(* IEC 61131-3 sources: verifaps-lib/geteta/examples/RTT_if (part 5) *)

        Pusher_states_t#Reset_interconnect_Slide1_Black:
             b_Pusher$_transit  := FALSE;
             b_Pusher$interconnect3  := FALSE;
             b_Pusher$Timer3$IN  := FALSE;
             b_Pusher$Timer3$PT  := USINT#0;
            IF  b_Pusher$Timer3$IN  THEN
                 b_Pusher$Timer3$Q  := ( b_Pusher$Timer3$ET  = USINT#0);
                IF ( b_Pusher$Timer3$ET  > USINT#0) THEN
                     b_Pusher$Timer3$ET  := ( b_Pusher$Timer3$ET  - USINT#1);
                ELSE
                     b_Pusher$Timer3$ET  := USINT#0;
                END_IF
            ELSE
                 b_Pusher$Timer3$Q  := FALSE;
                 b_Pusher$Timer3$ET  :=  b_Pusher$Timer3$PT ;
            END_IF
             b_Pusher$interconnect_Slide1_Black  := FALSE;
             b_Pusher$Timer_Slide1_Black$IN  := FALSE;
             b_Pusher$Timer_Slide1_Black$PT  := USINT#0;
            IF  b_Pusher$Timer_Slide1_Black$IN  THEN
                 b_Pusher$Timer_Slide1_Black$Q  := ( b_Pusher$Timer_Slide1_Black$ET  = USINT#0);
                IF ( b_Pusher$Timer_Slide1_Black$ET  > USINT#0) THEN
                     b_Pusher$Timer_Slide1_Black$ET  := ( b_Pusher$Timer_Slide1_Black$ET  - USINT#1);
                ELSE
                     b_Pusher$Timer_Slide1_Black$ET  := USINT#0;
                END_IF
            ELSE
                 b_Pusher$Timer_Slide1_Black$Q  := FALSE;
                 b_Pusher$Timer_Slide1_Black$ET  :=  b_Pusher$Timer_Slide1_Black$PT ;
            END_IF
             b_Pusher$Slide1_black  := ( b_Pusher$Slide1_black  - INT#1);
             b_Pusher$Priority_Var_Black  := ( b_Pusher$Priority_Var_Black  - INT#1);
            IF TRUE THEN
                 b_Pusher$_transit  := TRUE;
                 b_Pusher$_state  := Pusher_states_t#Interstep_2;
            END_IF

        Pusher_states_t#Reset_interconnect_Slide1_Metal:
             b_Pusher$_transit  := FALSE;
             b_Pusher$interconnect3  := FALSE;
             b_Pusher$Timer3$IN  := FALSE;
             b_Pusher$Timer3$PT  := USINT#0;
            IF  b_Pusher$Timer3$IN  THEN
                 b_Pusher$Timer3$Q  := ( b_Pusher$Timer3$ET  = USINT#0);
                IF ( b_Pusher$Timer3$ET  > USINT#0) THEN
                     b_Pusher$Timer3$ET  := ( b_Pusher$Timer3$ET  - USINT#1);
                ELSE
                     b_Pusher$Timer3$ET  := USINT#0;
                END_IF
            ELSE
                 b_Pusher$Timer3$Q  := FALSE;
                 b_Pusher$Timer3$ET  :=  b_Pusher$Timer3$PT ;
            END_IF
             b_Pusher$interconnect_Slide1_Metal  := FALSE;
             b_Pusher$Timer_Slide1_Metal$IN  := FALSE;
             b_Pusher$Timer_Slide1_Metal$PT  := USINT#0;
            IF  b_Pusher$Timer_Slide1_Metal$IN  THEN
                 b_Pusher$Timer_Slide1_Metal$Q  := ( b_Pusher$Timer_Slide1_Metal$ET  = USINT#0);
                IF ( b_Pusher$Timer_Slide1_Metal$ET  > USINT#0) THEN
                     b_Pusher$Timer_Slide1_Metal$ET  := ( b_Pusher$Timer_Slide1_Metal$ET  - USINT#1);
                ELSE
                     b_Pusher$Timer_Slide1_Metal$ET  := USINT#0;
                END_IF
            ELSE
                 b_Pusher$Timer_Slide1_Metal$Q  := FALSE;
                 b_Pusher$Timer_Slide1_Metal$ET  :=  b_Pusher$Timer_Slide1_Metal$PT ;
            END_IF
             b_Pusher$Slide1_metal  := ( b_Pusher$Slide1_metal  - INT#1);
             b_Pusher$Priority_Var_Metal  := ( b_Pusher$Priority_Var_Metal  - INT#1);
            IF TRUE THEN
                 b_Pusher$_transit  := TRUE;
                 b_Pusher$_state  := Pusher_states_t#Interstep_2;
            END_IF

        Pusher_states_t#Reset_interconnect_Slide1_White:
             b_Pusher$_transit  := FALSE;
             b_Pusher$interconnect3  := FALSE;
             b_Pusher$Timer3$IN  := FALSE;
             b_Pusher$Timer3$PT  := USINT#0;
            IF  b_Pusher$Timer3$IN  THEN
                 b_Pusher$Timer3$Q  := ( b_Pusher$Timer3$ET  = USINT#0);
                IF ( b_Pusher$Timer3$ET  > USINT#0) THEN
                     b_Pusher$Timer3$ET  := ( b_Pusher$Timer3$ET  - USINT#1);
                ELSE
                     b_Pusher$Timer3$ET  := USINT#0;
                END_IF
            ELSE
                 b_Pusher$Timer3$Q  := FALSE;
                 b_Pusher$Timer3$ET  :=  b_Pusher$Timer3$PT ;
            END_IF
             b_Pusher$interconnect_Slide1_White  := FALSE;
             b_Pusher$Timer_Slide1_White$IN  := FALSE;
             b_Pusher$Timer_Slide1_White$PT  := USINT#0;
            IF  b_Pusher$Timer_Slide1_White$IN  THEN
                 b_Pusher$Timer_Slide1_White$Q  := ( b_Pusher$Timer_Slide1_White$ET  = USINT#0);
                IF ( b_Pusher$Timer_Slide1_White$ET  > USINT#0) THEN
                     b_Pusher$Timer_Slide1_White$ET  := ( b_Pusher$Timer_Slide1_White$ET  - USINT#1);
                ELSE
                     b_Pusher$Timer_Slide1_White$ET  := USINT#0;
                END_IF
            ELSE
                 b_Pusher$Timer_Slide1_White$Q  := FALSE;
                 b_Pusher$Timer_Slide1_White$ET  :=  b_Pusher$Timer_Slide1_White$PT ;
            END_IF
             b_Pusher$Slide1_white  := ( b_Pusher$Slide1_white  - INT#1);
             b_Pusher$Priority_Var_White  := ( b_Pusher$Priority_Var_White  - INT#1);
            IF TRUE THEN
                 b_Pusher$_transit  := TRUE;
                 b_Pusher$_state  := Pusher_states_t#Interstep_2;
            END_IF

        Pusher_states_t#Reset_interconnect_Slide2_Black:
             b_Pusher$_transit  := FALSE;
             b_Pusher$interconnect3  := FALSE;
             b_Pusher$Timer3$IN  := FALSE;
             b_Pusher$Timer3$PT  := USINT#0;
            IF  b_Pusher$Timer3$IN  THEN
                 b_Pusher$Timer3$Q  := ( b_Pusher$Timer3$ET  = USINT#0);
                IF ( b_Pusher$Timer3$ET  > USINT#0) THEN
                     b_Pusher$Timer3$ET  := ( b_Pusher$Timer3$ET  - USINT#1);
                ELSE
                     b_Pusher$Timer3$ET  := USINT#0;
                END_IF
            ELSE
                 b_Pusher$Timer3$Q  := FALSE;
                 b_Pusher$Timer3$ET  :=  b_Pusher$Timer3$PT ;
            END_IF
             b_Pusher$interconnect_Slide2_Black  := FALSE;
             b_Pusher$Timer_Slide2_Black$IN  := FALSE;
             b_Pusher$Timer_Slide2_Black$PT  := USINT#0;
            IF  b_Pusher$Timer_Slide2_Black$IN  THEN
                 b_Pusher$Timer_Slide2_Black$Q  := ( b_Pusher$Timer_Slide2_Black$ET  = USINT#0);
                IF ( b_Pusher$Timer_Slide2_Black$ET  > USINT#0) THEN
                     b_Pusher$Timer_Slide2_Black$ET  := ( b_Pusher$Timer_Slide2_Black$ET  - USINT#1);
                ELSE
                     b_Pusher$Timer_Slide2_Black$ET  := USINT#0;
                END_IF
            ELSE
                 b_Pusher$Timer_Slide2_Black$Q  := FALSE;
                 b_Pusher$Timer_Slide2_Black$ET  :=  b_Pusher$Timer_Slide2_Black$PT ;
            END_IF
             b_Pusher$Slide2_black  := ( b_Pusher$Slide2_black  - INT#1);
             b_Pusher$Priority_Var_Black  := ( b_Pusher$Priority_Var_Black  - INT#1);
            IF TRUE THEN
                 b_Pusher$_transit  := TRUE;
                 b_Pusher$_state  := Pusher_states_t#Interstep_2;
            END_IF

        Pusher_states_t#Reset_interconnect_Slide2_Metal:
             b_Pusher$_transit  := FALSE;
             b_Pusher$interconnect3  := FALSE;
             b_Pusher$Timer3$IN  := FALSE;
             b_Pusher$Timer3$PT  := USINT#0;
            IF  b_Pusher$Timer3$IN  THEN
                 b_Pusher$Timer3$Q  := ( b_Pusher$Timer3$ET  = USINT#0);
                IF ( b_Pusher$Timer3$ET  > USINT#0) THEN
                     b_Pusher$Timer3$ET  := ( b_Pusher$Timer3$ET  - USINT#1);
                ELSE
                     b_Pusher$Timer3$ET  := USINT#0;
                END_IF
            ELSE
                 b_Pusher$Timer3$Q  := FALSE;
                 b_Pusher$Timer3$ET  :=  b_Pusher$Timer3$PT ;
            END_IF
             b_Pusher$interconnect_Slide2_Metal  := FALSE;
             b_Pusher$Timer_Slide2_Metal$IN  := FALSE;
             b_Pusher$Timer_Slide2_Metal$PT  := USINT#0;
            IF  b_Pusher$Timer_Slide2_Metal$IN  THEN
                 b_Pusher$Timer_Slide2_Metal$Q  := ( b_Pusher$Timer_Slide2_Metal$ET  = USINT#0);
                IF ( b_Pusher$Timer_Slide2_Metal$ET  > USINT#0) THEN
                     b_Pusher$Timer_Slide2_Metal$ET  := ( b_Pusher$Timer_Slide2_Metal$ET  - USINT#1);
                ELSE
                     b_Pusher$Timer_Slide2_Metal$ET  := USINT#0;
                END_IF
            ELSE
                 b_Pusher$Timer_Slide2_Metal$Q  := FALSE;
                 b_Pusher$Timer_Slide2_Metal$ET  :=  b_Pusher$Timer_Slide2_Metal$PT ;
            END_IF
             b_Pusher$Slide2_metal  := ( b_Pusher$Slide2_metal  - INT#1);
             b_Pusher$Priority_Var_Metal  := ( b_Pusher$Priority_Var_Metal  - INT#1);
            IF TRUE THEN
                 b_Pusher$_transit  := TRUE;
                 b_Pusher$_state  := Pusher_states_t#Interstep_2;
            END_IF

        Pusher_states_t#Reset_interconnect_Slide2_White:
             b_Pusher$_transit  := FALSE;
             b_Pusher$interconnect3  := FALSE;
             b_Pusher$Timer3$IN  := FALSE;
             b_Pusher$Timer3$PT  := USINT#0;
            IF  b_Pusher$Timer3$IN  THEN
                 b_Pusher$Timer3$Q  := ( b_Pusher$Timer3$ET  = USINT#0);
                IF ( b_Pusher$Timer3$ET  > USINT#0) THEN
                     b_Pusher$Timer3$ET  := ( b_Pusher$Timer3$ET  - USINT#1);
                ELSE
                     b_Pusher$Timer3$ET  := USINT#0;
                END_IF
            ELSE
                 b_Pusher$Timer3$Q  := FALSE;
                 b_Pusher$Timer3$ET  :=  b_Pusher$Timer3$PT ;
            END_IF
             b_Pusher$interconnect_Slide2_White  := FALSE;
             b_Pusher$Timer_Slide2_White$IN  := FALSE;
             b_Pusher$Timer_Slide2_White$PT  := USINT#0;
            IF  b_Pusher$Timer_Slide2_White$IN  THEN
                 b_Pusher$Timer_Slide2_White$Q  := ( b_Pusher$Timer_Slide2_White$ET  = USINT#0);
                IF ( b_Pusher$Timer_Slide2_White$ET  > USINT#0) THEN
                     b_Pusher$Timer_Slide2_White$ET  := ( b_Pusher$Timer_Slide2_White$ET  - USINT#1);
                ELSE
                     b_Pusher$Timer_Slide2_White$ET  := USINT#0;
                END_IF
            ELSE
                 b_Pusher$Timer_Slide2_White$Q  := FALSE;
                 b_Pusher$Timer_Slide2_White$ET  :=  b_Pusher$Timer_Slide2_White$PT ;
            END_IF
             b_Pusher$Slide2_white  := ( b_Pusher$Slide2_white  - INT#1);
             b_Pusher$Priority_Var_White  := ( b_Pusher$Priority_Var_White  - INT#1);
            IF TRUE THEN
                 b_Pusher$_transit  := TRUE;
                 b_Pusher$_state  := Pusher_states_t#Interstep_2;
            END_IF

        Pusher_states_t#Reset_interconnect_Slide3_Metal:
             b_Pusher$_transit  := FALSE;
             b_Pusher$interconnect3  := FALSE;
             b_Pusher$Timer3$IN  := FALSE;
             b_Pusher$Timer3$PT  := USINT#0;
            IF  b_Pusher$Timer3$IN  THEN
                 b_Pusher$Timer3$Q  := ( b_Pusher$Timer3$ET  = USINT#0);
                IF ( b_Pusher$Timer3$ET  > USINT#0) THEN
                     b_Pusher$Timer3$ET  := ( b_Pusher$Timer3$ET  - USINT#1);
                ELSE
                     b_Pusher$Timer3$ET  := USINT#0;
                END_IF
            ELSE
                 b_Pusher$Timer3$Q  := FALSE;
                 b_Pusher$Timer3$ET  :=  b_Pusher$Timer3$PT ;
            END_IF
             b_Pusher$Slide3_metal  := ( b_Pusher$Slide3_metal  - INT#1);
             b_Pusher$Priority_Var_Metal  := ( b_Pusher$Priority_Var_Metal  - INT#1);
            IF TRUE THEN
                 b_Pusher$_transit  := TRUE;
                 b_Pusher$_state  := Pusher_states_t#Interstep_2;
            END_IF

        Pusher_states_t#Reset_interconnect_Slide3_White:
             b_Pusher$_transit  := FALSE;
             b_Pusher$interconnect3  := FALSE;
             b_Pusher$Timer3$IN  := FALSE;
             b_Pusher$Timer3$PT  := USINT#0;
            IF  b_Pusher$Timer3$IN  THEN
                 b_Pusher$Timer3$Q  := ( b_Pusher$Timer3$ET  = USINT#0);
                IF ( b_Pusher$Timer3$ET  > USINT#0) THEN
                     b_Pusher$Timer3$ET  := ( b_Pusher$Timer3$ET  - USINT#1);
                ELSE
                     b_Pusher$Timer3$ET  := USINT#0;
                END_IF
            ELSE
                 b_Pusher$Timer3$Q  := FALSE;
                 b_Pusher$Timer3$ET  :=  b_Pusher$Timer3$PT ;
            END_IF
             b_Pusher$Slide3_white  := ( b_Pusher$Slide3_white  - INT#1);
             b_Pusher$Priority_Var_White  := ( b_Pusher$Priority_Var_White  - INT#1);
            IF TRUE THEN
                 b_Pusher$_transit  := TRUE;
                 b_Pusher$_state  := Pusher_states_t#Interstep_2;
            END_IF

        Pusher_states_t#Second_Slide_Timer_Black:
             b_Pusher$_transit  := FALSE;
            IF ( b_Pusher$SorterLightnesssensorCraneInterfaceInverse  = TRUE) THEN
                 b_Pusher$Timer_Slide2_Black$IN  :=  b_Pusher$SorterLightnesssensorCraneInterfaceInverse ;
                 b_Pusher$Timer_Slide2_Black$PT  :=  b_Pusher$Duration_Slide2_Black ;
                IF  b_Pusher$Timer_Slide2_Black$IN  THEN
                     b_Pusher$Timer_Slide2_Black$Q  := ( b_Pusher$Timer_Slide2_Black$ET  = USINT#0);
                    IF ( b_Pusher$Timer_Slide2_Black$ET  > USINT#0) THEN
                         b_Pusher$Timer_Slide2_Black$ET  := ( b_Pusher$Timer_Slide2_Black$ET  - USINT#1);
                    ELSE
                         b_Pusher$Timer_Slide2_Black$ET  := USINT#0;
                    END_IF
                ELSE
                     b_Pusher$Timer_Slide2_Black$Q  := FALSE;
                     b_Pusher$Timer_Slide2_Black$ET  :=  b_Pusher$Timer_Slide2_Black$PT ;
                END_IF
                 b_Pusher$interconnect_Slide2_Black  :=  b_Pusher$Timer_Slide2_Black$Q ;
            END_IF
            IF  b_Pusher$interconnect_Slide2_Black  THEN
                 b_Pusher$_transit  := TRUE;
                 b_Pusher$_state  := Pusher_states_t#PusherY2_Move_Out_Black;
            END_IF

        Pusher_states_t#Second_Slide_Timer_Metal:
             b_Pusher$_transit  := FALSE;
             b_Pusher$Timer_Slide2_Metal$IN  := TRUE;
             b_Pusher$Timer_Slide2_Metal$PT  :=  b_Pusher$Duration_Slide2_Metal ;
            IF  b_Pusher$Timer_Slide2_Metal$IN  THEN
                 b_Pusher$Timer_Slide2_Metal$Q  := ( b_Pusher$Timer_Slide2_Metal$ET  = USINT#0);
                IF ( b_Pusher$Timer_Slide2_Metal$ET  > USINT#0) THEN
                     b_Pusher$Timer_Slide2_Metal$ET  := ( b_Pusher$Timer_Slide2_Metal$ET  - USINT#1);
                ELSE
                     b_Pusher$Timer_Slide2_Metal$ET  := USINT#0;
                END_IF
            ELSE
                 b_Pusher$Timer_Slide2_Metal$Q  := FALSE;
                 b_Pusher$Timer_Slide2_Metal$ET  :=  b_Pusher$Timer_Slide2_Metal$PT ;
            END_IF
             b_Pusher$interconnect_Slide2_Metal  :=  b_Pusher$Timer_Slide2_Metal$Q ;
            IF  b_Pusher$interconnect_Slide2_Metal  THEN
                 b_Pusher$_transit  := TRUE;
                 b_Pusher$_state  := Pusher_states_t#PusherY2_Move_Out_Metal;
            END_IF

        Pusher_states_t#Second_Slide_Timer_White:
             b_Pusher$_transit  := FALSE;
             b_Pusher$Timer_Slide2_White$IN  := TRUE;
             b_Pusher$Timer_Slide2_White$PT  :=  b_Pusher$Duration_Slide2_White ;
            IF  b_Pusher$Timer_Slide2_White$IN  THEN
                 b_Pusher$Timer_Slide2_White$Q  := ( b_Pusher$Timer_Slide2_White$ET  = USINT#0);
                IF ( b_Pusher$Timer_Slide2_White$ET  > USINT#0) THEN
                     b_Pusher$Timer_Slide2_White$ET  := ( b_Pusher$Timer_Slide2_White$ET  - USINT#1);
                ELSE
                     b_Pusher$Timer_Slide2_White$ET  := USINT#0;
                END_IF
            ELSE
                 b_Pusher$Timer_Slide2_White$Q  := FALSE;
                 b_Pusher$Timer_Slide2_White$ET  :=  b_Pusher$Timer_Slide2_White$PT ;
            END_IF
             b_Pusher$interconnect_Slide2_White  :=  b_Pusher$Timer_Slide2_White$Q ;
            IF  b_Pusher$interconnect_Slide2_White  THEN
                 b_Pusher$_transit  := TRUE;
                 b_Pusher$_state  := Pusher_states_t#PusherY2_Move_Out_White;
            END_IF

        Pusher_states_t#Second_Slide_black_workpieces:
             b_Pusher$_transit  := FALSE;
            IF TRUE THEN
                 b_Pusher$_transit  := TRUE;
                 b_Pusher$_state  := Pusher_states_t#Second_Slide_Timer_Black;
            END_IF

        Pusher_states_t#Second_Slide_metal_workpieces:
             b_Pusher$_transit  := FALSE;
            IF ( b_Pusher$SorterLightnessSensorPusher2  AND  b_Pusher$SorterCapacitiveSensorPusher2 ) THEN
                 b_Pusher$_transit  := TRUE;
                 b_Pusher$_state  := Pusher_states_t#Second_Test_For_Metal;
            END_IF

        Pusher_states_t#Second_Slide_white_workpieces:
             b_Pusher$_transit  := FALSE;
            IF ( b_Pusher$SorterLightnessSensorPusher2  AND NOT  b_Pusher$SorterCapacitiveSensorPusher2 ) THEN
                 b_Pusher$_transit  := TRUE;
                 b_Pusher$_state  := Pusher_states_t#Second_Test_For_White;
            END_IF

        Pusher_states_t#Second_Test_For_Metal:
             b_Pusher$_transit  := FALSE;
            IF TRUE THEN
                 b_Pusher$_transit  := TRUE;
                 b_Pusher$_state  := Pusher_states_t#Second_Slide_Timer_Metal;
            END_IF

        Pusher_states_t#Second_Test_For_White:
             b_Pusher$_transit  := FALSE;
            IF TRUE THEN
                 b_Pusher$_transit  := TRUE;
                 b_Pusher$_state  := Pusher_states_t#Second_Slide_Timer_White;
            END_IF

        Pusher_states_t#Third_Slide_black_workpieces:
             b_Pusher$_transit  := FALSE;
            IF (NOT  b_Pusher$SorterLightnessSensorPusher2  AND NOT  b_Pusher$SorterCapacitiveSensorPusher2 ) THEN
                 b_Pusher$_transit  := TRUE;
                 b_Pusher$_state  := Pusher_states_t#Wait_Black;
            END_IF

        Pusher_states_t#Third_Slide_metal_workpieces:
             b_Pusher$_transit  := FALSE;
            IF ( b_Pusher$SorterLightnessSensorPusher2  AND  b_Pusher$SorterCapacitiveSensorPusher2 ) THEN
                 b_Pusher$_transit  := TRUE;
                 b_Pusher$_state  := Pusher_states_t#Wait_Metal;
            END_IF

        Pusher_states_t#Third_Slide_white_workpieces:
             b_Pusher$_transit  := FALSE;
            IF ( b_Pusher$SorterLightnessSensorPusher2  AND NOT  b_Pusher$SorterCapacitiveSensorPusher2 ) THEN
                 b_Pusher$_transit  := TRUE;
                 b_Pusher$_state  := Pusher_states_t#Wait_White;
            END_IF

        Pusher_states_t#Wait_Black:
             b_Pusher$_transit  := FALSE;
            IF ((NOT  b_Pusher$SorterLightnessSensorPusher2  AND NOT  b_Pusher$SorterCapacitiveSensorPusher2 ) = TRUE) THEN
                 b_Pusher$Timer2$IN  := (NOT  b_Pusher$SorterLightnessSensorPusher2  AND NOT  b_Pusher$SorterCapacitiveSensorPusher2 );
                 b_Pusher$Timer2$PT  :=  b_Pusher$Duration2 ;
                IF  b_Pusher$Timer2$IN  THEN
                     b_Pusher$Timer2$Q  := ( b_Pusher$Timer2$ET  = USINT#0);
                    IF ( b_Pusher$Timer2$ET  > USINT#0) THEN
                         b_Pusher$Timer2$ET  := ( b_Pusher$Timer2$ET  - USINT#1);
                    ELSE
                         b_Pusher$Timer2$ET  := USINT#0;
                    END_IF
                ELSE
                     b_Pusher$Timer2$Q  := FALSE;
                     b_Pusher$Timer2$ET  :=  b_Pusher$Timer2$PT ;
                END_IF
                 b_Pusher$interconnect2  :=  b_Pusher$Timer2$Q ;
            END_IF
            IF  b_Pusher$interconnect2  THEN
                 b_Pusher$_transit  := TRUE;
                 b_Pusher$_state  := Pusher_states_t#Reset_interconnect3;
            END_IF

        Pusher_states_t#Wait_Metal:
             b_Pusher$_transit  := FALSE;
             b_Pusher$Timer3$IN  := TRUE;
             b_Pusher$Timer3$PT  :=  b_Pusher$Duration3 ;
            IF  b_Pusher$Timer3$IN  THEN
                 b_Pusher$Timer3$Q  := ( b_Pusher$Timer3$ET  = USINT#0);
                IF ( b_Pusher$Timer3$ET  > USINT#0) THEN
                     b_Pusher$Timer3$ET  := ( b_Pusher$Timer3$ET  - USINT#1);
                ELSE
                     b_Pusher$Timer3$ET  := USINT#0;
                END_IF
            ELSE
                 b_Pusher$Timer3$Q  := FALSE;
                 b_Pusher$Timer3$ET  :=  b_Pusher$Timer3$PT ;
            END_IF
             b_Pusher$interconnect3  :=  b_Pusher$Timer3$Q ;
            IF  b_Pusher$interconnect3  THEN
                 b_Pusher$_transit  := TRUE;
                 b_Pusher$_state  := Pusher_states_t#Reset_interconnect_Slide3_Metal;
            END_IF

        Pusher_states_t#Wait_White:
             b_Pusher$_transit  := FALSE;
             b_Pusher$Timer3$IN  := TRUE;
             b_Pusher$Timer3$PT  :=  b_Pusher$Duration3 ;
            IF  b_Pusher$Timer3$IN  THEN
                 b_Pusher$Timer3$Q  := ( b_Pusher$Timer3$ET  = USINT#0);
                IF ( b_Pusher$Timer3$ET  > USINT#0) THEN
                     b_Pusher$Timer3$ET  := ( b_Pusher$Timer3$ET  - USINT#1);
                ELSE
                     b_Pusher$Timer3$ET  := USINT#0;
                END_IF
            ELSE
                 b_Pusher$Timer3$Q  := FALSE;
                 b_Pusher$Timer3$ET  :=  b_Pusher$Timer3$PT ;
            END_IF
             b_Pusher$interconnect3  :=  b_Pusher$Timer3$Q ;
            IF  b_Pusher$interconnect3  THEN
                 b_Pusher$_transit  := TRUE;
                 b_Pusher$_state  := Pusher_states_t#Reset_interconnect_Slide3_White;
            END_IF

        Pusher_states_t#Wait_Y1_Black:
             b_Pusher$_transit  := FALSE;
            IF ( b_Pusher$PusherY1  = TRUE) THEN
                 b_Pusher$Timer3$IN  :=  b_Pusher$PusherY1 ;
                 b_Pusher$Timer3$PT  :=  b_Pusher$Duration3 ;
                IF  b_Pusher$Timer3$IN  THEN
                     b_Pusher$Timer3$Q  := ( b_Pusher$Timer3$ET  = USINT#0);
                    IF ( b_Pusher$Timer3$ET  > USINT#0) THEN
                         b_Pusher$Timer3$ET  := ( b_Pusher$Timer3$ET  - USINT#1);
                    ELSE
                         b_Pusher$Timer3$ET  := USINT#0;
                    END_IF
                ELSE
                     b_Pusher$Timer3$Q  := FALSE;
                     b_Pusher$Timer3$ET  :=  b_Pusher$Timer3$PT ;
                END_IF
                 b_Pusher$interconnect3  :=  b_Pusher$Timer3$Q ;
            END_IF
            IF  b_Pusher$interconnect3  THEN
                 b_Pusher$_transit  := TRUE;
                 b_Pusher$_state  := Pusher_states_t#PusherY1_Move_In_Black;
            END_IF

        Pusher_states_t#Wait_Y1_Metal:
             b_Pusher$_transit  := FALSE;
            IF ( b_Pusher$PusherY1  = TRUE) THEN
                 b_Pusher$Timer3$IN  :=  b_Pusher$PusherY1 ;
                 b_Pusher$Timer3$PT  :=  b_Pusher$Duration3 ;
                IF  b_Pusher$Timer3$IN  THEN
                     b_Pusher$Timer3$Q  := ( b_Pusher$Timer3$ET  = USINT#0);
                    IF ( b_Pusher$Timer3$ET  > USINT#0) THEN
                         b_Pusher$Timer3$ET  := ( b_Pusher$Timer3$ET  - USINT#1);
                    ELSE
                         b_Pusher$Timer3$ET  := USINT#0;
                    END_IF
                ELSE
                     b_Pusher$Timer3$Q  := FALSE;
                     b_Pusher$Timer3$ET  :=  b_Pusher$Timer3$PT ;
                END_IF
                 b_Pusher$interconnect3  :=  b_Pusher$Timer3$Q ;
            END_IF
            IF  b_Pusher$interconnect3  THEN
                 b_Pusher$_transit  := TRUE;
                 b_Pusher$_state  := Pusher_states_t#PusherY1_Move_In_Metal;
            END_IF

        Pusher_states_t#Wait_Y1_White:
             b_Pusher$_transit  := FALSE;
            IF ( b_Pusher$PusherY1  = TRUE) THEN
                 b_Pusher$Timer3$IN  :=  b_Pusher$PusherY1 ;
                 b_Pusher$Timer3$PT  :=  b_Pusher$Duration3 ;
                IF  b_Pusher$Timer3$IN  THEN
                     b_Pusher$Timer3$Q  := ( b_Pusher$Timer3$ET  = USINT#0);
                    IF ( b_Pusher$Timer3$ET  > USINT#0) THEN
                         b_Pusher$Timer3$ET  := ( b_Pusher$Timer3$ET  - USINT#1);
                    ELSE
                         b_Pusher$Timer3$ET  := USINT#0;
                    END_IF
                ELSE
                     b_Pusher$Timer3$Q  := FALSE;
                     b_Pusher$Timer3$ET  :=  b_Pusher$Timer3$PT ;
                END_IF
                 b_Pusher$interconnect3  :=  b_Pusher$Timer3$Q ;
            END_IF
            IF  b_Pusher$interconnect3  THEN
                 b_Pusher$_transit  := TRUE;
                 b_Pusher$_state  := Pusher_states_t#PusherY1_Move_In_White;
            END_IF

        Pusher_states_t#Wait_Y2_Black:
             b_Pusher$_transit  := FALSE;
            IF ( b_Pusher$PusherY2  = TRUE) THEN
                 b_Pusher$Timer3$IN  :=  b_Pusher$PusherY2 ;
                 b_Pusher$Timer3$PT  :=  b_Pusher$Duration3 ;
                IF  b_Pusher$Timer3$IN  THEN
                     b_Pusher$Timer3$Q  := ( b_Pusher$Timer3$ET  = USINT#0);
                    IF ( b_Pusher$Timer3$ET  > USINT#0) THEN
                         b_Pusher$Timer3$ET  := ( b_Pusher$Timer3$ET  - USINT#1);
                    ELSE
                         b_Pusher$Timer3$ET  := USINT#0;
                    END_IF
                ELSE
                     b_Pusher$Timer3$Q  := FALSE;
                     b_Pusher$Timer3$ET  :=  b_Pusher$Timer3$PT ;
                END_IF
                 b_Pusher$interconnect3  :=  b_Pusher$Timer3$Q ;
            END_IF
            IF  b_Pusher$interconnect3  THEN
                 b_Pusher$_transit  := TRUE;
                 b_Pusher$_state  := Pusher_states_t#PusherY2_Move_In_Black;
            END_IF

        Pusher_states_t#Wait_Y2_Metal:
             b_Pusher$_transit  := FALSE;
            IF ( b_Pusher$PusherY2  = TRUE) THEN
                 b_Pusher$Timer3$IN  :=  b_Pusher$PusherY2 ;
                 b_Pusher$Timer3$PT  :=  b_Pusher$Duration3 ;
                IF  b_Pusher$Timer3$IN  THEN
                     b_Pusher$Timer3$Q  := ( b_Pusher$Timer3$ET  = USINT#0);
                    IF ( b_Pusher$Timer3$ET  > USINT#0) THEN
                         b_Pusher$Timer3$ET  := ( b_Pusher$Timer3$ET  - USINT#1);
                    ELSE
                         b_Pusher$Timer3$ET  := USINT#0;
                    END_IF
                ELSE
                     b_Pusher$Timer3$Q  := FALSE;
                     b_Pusher$Timer3$ET  :=  b_Pusher$Timer3$PT ;
                END_IF
                 b_Pusher$interconnect3  :=  b_Pusher$Timer3$Q ;
            END_IF
            IF  b_Pusher$interconnect3  THEN
                 b_Pusher$_transit  := TRUE;
                 b_Pusher$_state  := Pusher_states_t#PusherY2_Move_In_Metal;
            END_IF

        Pusher_states_t#Wait_Y2_White:
             b_Pusher$_transit  := FALSE;
            IF ( b_Pusher$PusherY2  = TRUE) THEN
                 b_Pusher$Timer3$IN  :=  b_Pusher$PusherY2 ;
                 b_Pusher$Timer3$PT  :=  b_Pusher$Duration3 ;
                IF  b_Pusher$Timer3$IN  THEN
                     b_Pusher$Timer3$Q  := ( b_Pusher$Timer3$ET  = USINT#0);
                    IF ( b_Pusher$Timer3$ET  > USINT#0) THEN
                         b_Pusher$Timer3$ET  := ( b_Pusher$Timer3$ET  - USINT#1);
                    ELSE
                         b_Pusher$Timer3$ET  := USINT#0;
                    END_IF
                ELSE
                     b_Pusher$Timer3$Q  := FALSE;
                     b_Pusher$Timer3$ET  :=  b_Pusher$Timer3$PT ;
                END_IF
                 b_Pusher$interconnect3  :=  b_Pusher$Timer3$Q ;
            END_IF
            IF  b_Pusher$interconnect3  THEN
                 b_Pusher$_transit  := TRUE;
                 b_Pusher$_state  := Pusher_states_t#PusherY2_Move_In_White;
            END_IF

            END_CASE
    IF (( b_Actuator_SorterGreenLampConveyor  AND  b_Actuator_MagazinGreenLamp ) AND  b_Actuator_StampGreenLamp ) THEN
        IF ((( b_Stamp$StartCommandStamp  AND  b_Crane$StartCommandCrane ) AND  b_Conveyor$StartCommandConveyor ) AND  b_Mag$StartCommandMagazin ) THEN
             b_Crane$StartVar  := TRUE;
             b_Conveyor$StartVar  := TRUE;
             b_Mag$StartVar  := TRUE;
             b_Pusher$StartVar  := TRUE;
             b_Stamp$StartVar  := TRUE;
             b_DIAGNOSIS_ACTIVE  := TRUE;
        END_IF
    END_IF
     b_Crane$SFCReset  := FALSE;
     b_Conveyor$SFCReset  := FALSE;
     b_Mag$SFCReset  := FALSE;
     b_Pusher$SFCReset  := FALSE;
     b_Stamp$SFCReset  := FALSE;

     b_Crane$AnalogCranePressure  :=  b_PARAMETER_CRANE_PRESSURE_METALLIC ;

ELSEIF ((NOT  b_Sensor_SorterEmergencyStop  OR NOT  b_Sensor_StampEmergencyStop ) OR NOT  b_Sensor_MagazinEmergencyStop ) THEN
     b_Actuator_MagazinSlider  := FALSE;
     b_Actuator_CraneLower  := FALSE;
     b_Actuator_MagazinVacuumOn  := FALSE;
     b_Actuator_MagazinVacuumOff  := TRUE;
     b_Actuator_MagazinGreenLamp  := FALSE;
     b_Actuator_CraneTurnCounterclockwise  := FALSE;
     b_Actuator_CraneTurnClockwise  := FALSE;
     b_Actuator_SorterConveyorTowardsStacker  := FALSE;
     b_Actuator_SorterConveyorTowardsCrane  := FALSE;
     b_Actuator_SorterGreenLampConveyor  := FALSE;
     b_Actuator_PusherY1  := FALSE;
     b_Actuator_PusherY2  := FALSE;
     b_Actuator_StampSliderMovedOut  := TRUE;
     b_Actuator_StampSliderMovedIn  := FALSE;
     b_Actuator_StampGreenLamp  := FALSE;
     b_Actuator_StampPusher  := FALSE;
     b_Actuator_AnalogCranePressure  := INT#0;
     b_Crane$SFCReset  := TRUE;
     b_Conveyor$SFCReset  := TRUE;
     b_Mag$SFCReset  := TRUE;
     b_Pusher$SFCReset  := TRUE;
     b_Stamp$SFCReset  := TRUE;
     b_Crane$StartVar  := FALSE;
     b_Conveyor$StartVar  := FALSE;
     b_Mag$StartVar  := FALSE;
     b_Pusher$StartVar  := FALSE;
     b_Stamp$StartVar  := FALSE;
END_IF

 END_PROGRAM
